// TIA Portal V20 export
DATA_BLOCK "Simulation_DB"   // DB143
// stored: InstanceOfName Unit1.Em7.Simulation, InstanceOfType FB, Namespace Unit1.Em7
"Unit1.Em7.Simulation"
   // VAR
   //    Simulation_addon_Instance { S7_SetPoint := 'True'} : "Simulation_addon";
   //    statPulse : Bool;
   // END_VAR
BEGIN
END_DATA_BLOCK
